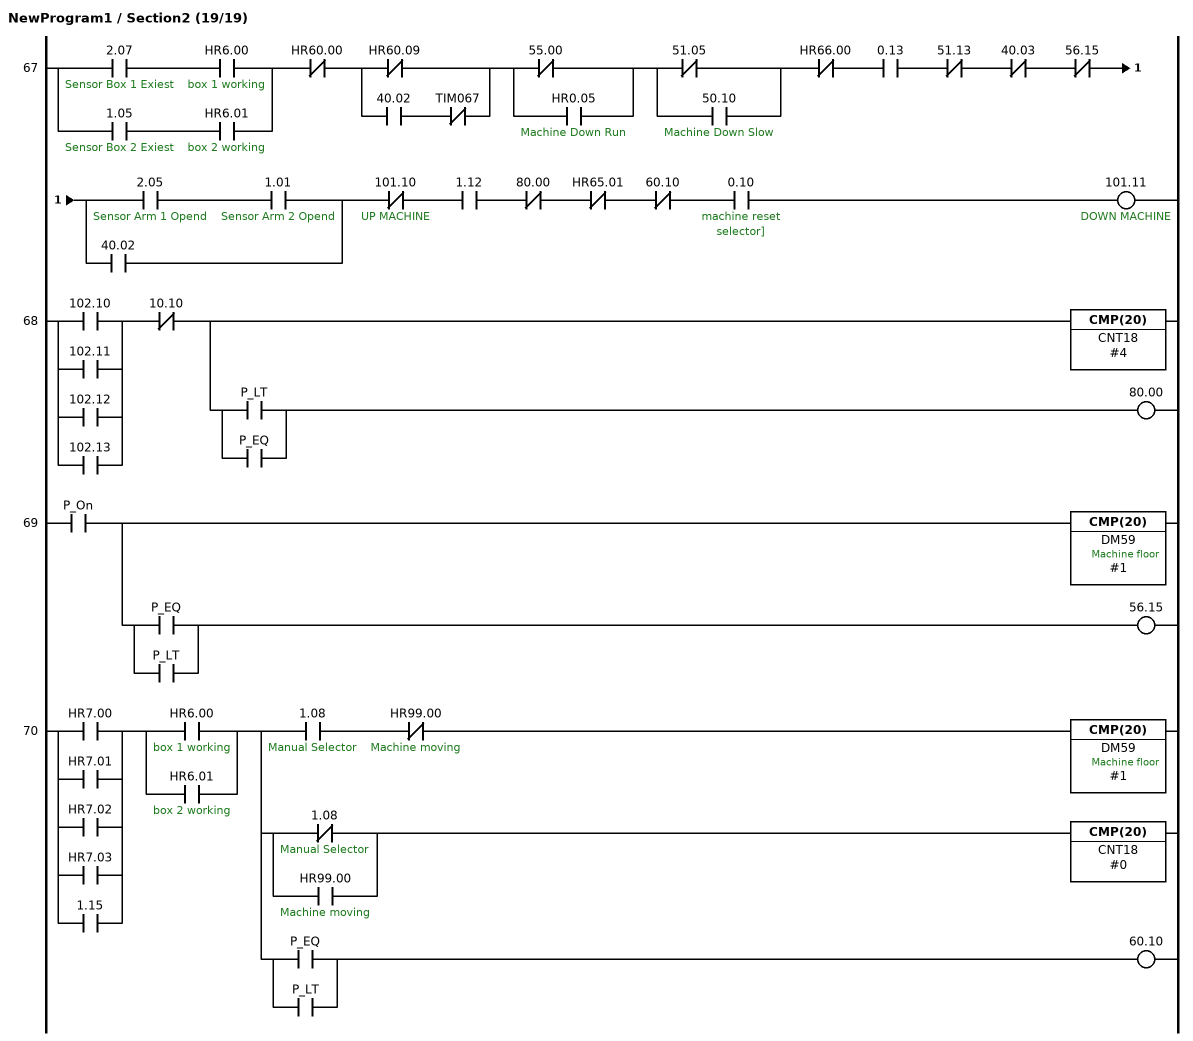
; [picture p24: NewProgram1 / Section2, rungs 67-70]
; rung 67
LD 2.07  ; Sensor Box 1 Exiest
AND HR6.00  ; box 1 working
LD 1.05  ; Sensor Box 2 Exiest
AND HR6.01  ; box 2 working
ORLD
ANDNOT HR60.00
LDNOT HR60.09
LD 40.02
ANDNOT TIM067
ORLD
ANDLD
LDNOT 55.00
OR HR0.05  ; Machine Down Run
ANDLD
LDNOT 51.05
OR 50.10  ; Machine Down Slow
ANDLD
ANDNOT HR66.00
AND 0.13
ANDNOT 51.13
ANDNOT 40.03
ANDNOT 56.15
LD 2.05  ; Sensor Arm 1 Opend
AND 1.01  ; Sensor Arm 2 Opend
OR 40.02
ANDLD
ANDNOT 101.10  ; UP MACHINE
AND 1.12
ANDNOT 80.00
ANDNOT HR65.01
ANDNOT 60.10
AND 0.10  ; machine reset selector]
OUT 101.11  ; DOWN MACHINE
; rung 68
LD 102.10
OR 102.11
OR 102.12
OR 102.13
ANDNOT 10.10
CMP(20) CNT18 #4
LD P_LT
OR P_EQ
ANDLD
OUT 80.00
; rung 69
LD P_On
CMP(20) DM59 #1  ; Machine floor
LD P_EQ
OR P_LT
ANDLD
OUT 56.15
; rung 70
LD HR7.00
OR HR7.01
OR HR7.02
OR HR7.03
OR 1.15
LD HR6.00  ; box 1 working
OR HR6.01  ; box 2 working
ANDLD
OUT TR0
AND 1.08  ; Manual Selector
ANDNOT HR99.00  ; Machine moving
CMP(20) DM59 #1  ; Machine floor
LD TR0
LDNOT 1.08  ; Manual Selector
OR HR99.00  ; Machine moving
ANDLD
CMP(20) CNT18 #0
LD TR0
LD P_EQ
OR P_LT
ANDLD
OUT 60.10

### Section Section3

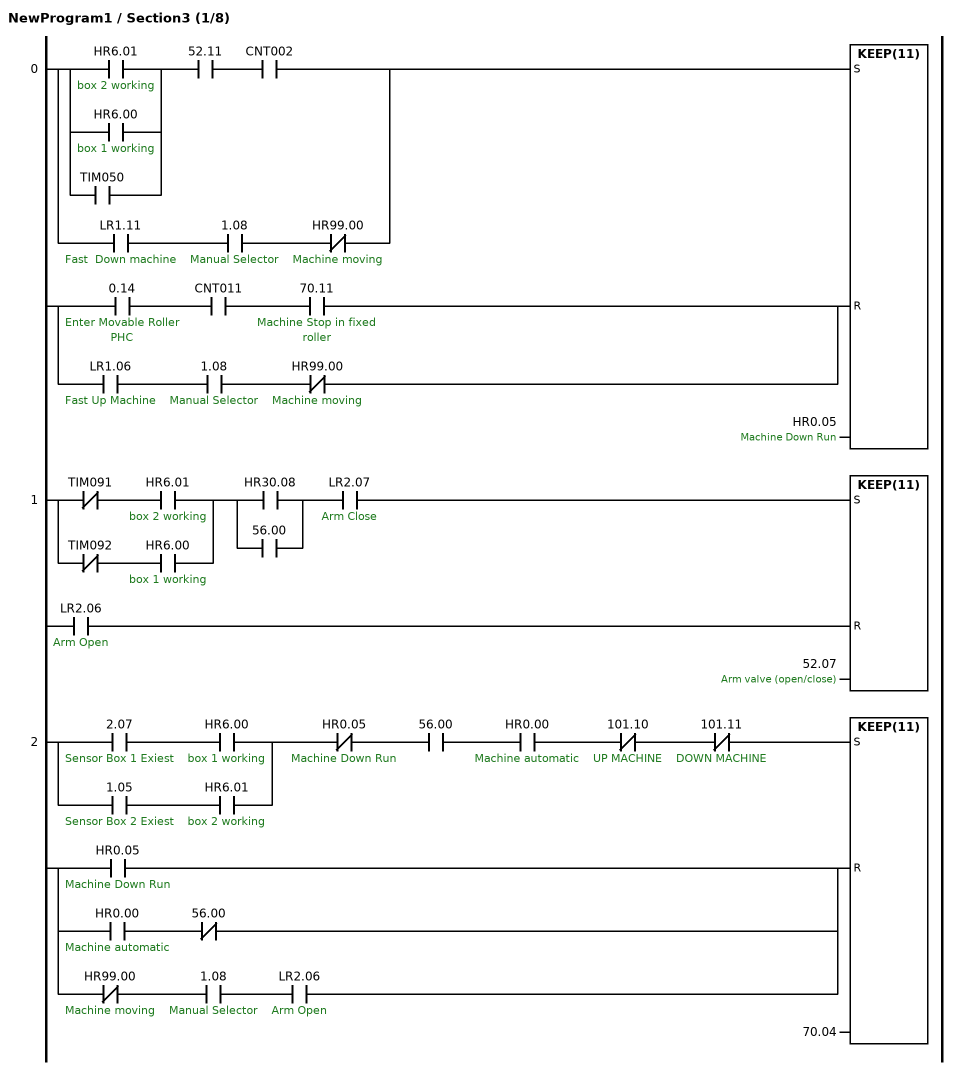
; rung 0
LD HR6.01  ; box 2 working
OR HR6.00  ; box 1 working
OR TIM050
AND 52.11
AND CNT002
LD LR1.11  ; Fast  Down machine
AND 1.08  ; Manual Selector
ANDNOT HR99.00  ; Machine moving
ORLD
LD 0.14  ; Enter Movable Roller PHC
AND CNT011
AND 70.11  ; Machine Stop in fixed roller
LD LR1.06  ; Fast Up Machine
AND 1.08  ; Manual Selector
ANDNOT HR99.00  ; Machine moving
ORLD
KEEP(11) HR0.05  ; Machine Down Run
; rung 1
LDNOT TIM091
AND HR6.01  ; box 2 working
LDNOT TIM092
AND HR6.00  ; box 1 working
ORLD
LD HR30.08
OR 56.00
ANDLD
AND LR2.07  ; Arm Close
LD LR2.06  ; Arm Open
KEEP(11) 52.07  ; Arm valve (open/close)
; rung 2
LD 2.07  ; Sensor Box 1 Exiest
AND HR6.00  ; box 1 working
LD 1.05  ; Sensor Box 2 Exiest
AND HR6.01  ; box 2 working
ORLD
ANDNOT HR0.05  ; Machine Down Run
AND 56.00
AND HR0.00  ; Machine automatic
ANDNOT 101.10  ; UP MACHINE
ANDNOT 101.11  ; DOWN MACHINE
LD HR0.05  ; Machine Down Run
LD HR0.00  ; Machine automatic
ANDNOT 56.00
ORLD
LDNOT HR99.00  ; Machine moving
AND 1.08  ; Manual Selector
AND LR2.06  ; Arm Open
ORLD
KEEP(11) 70.04

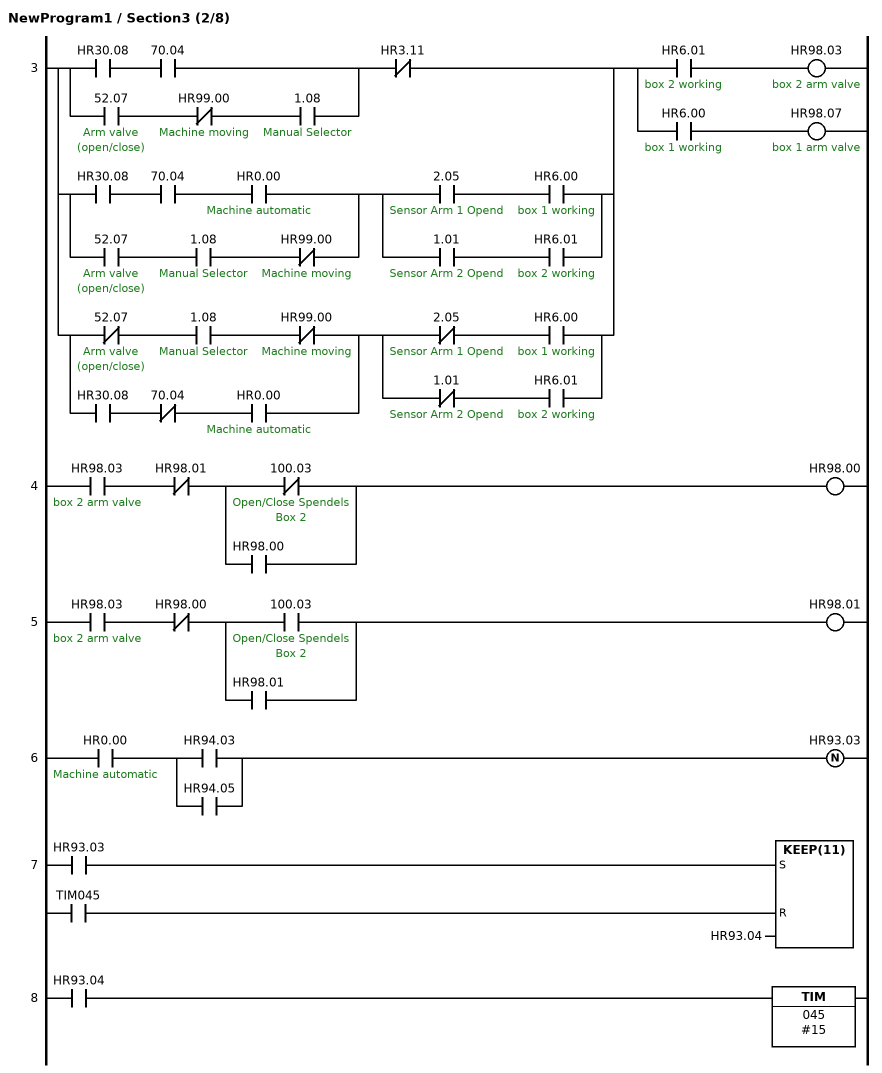
; rung 3
LD HR30.08
AND 70.04
LD 52.07  ; Arm valve (open/close)
ANDNOT HR99.00  ; Machine moving
AND 1.08  ; Manual Selector
ORLD
ANDNOT HR3.11
LD HR30.08
AND 70.04
AND HR0.00  ; Machine automatic
LD 52.07  ; Arm valve (open/close)
AND 1.08  ; Manual Selector
ANDNOT HR99.00  ; Machine moving
ORLD
LD 2.05  ; Sensor Arm 1 Opend
AND HR6.00  ; box 1 working
LD 1.01  ; Sensor Arm 2 Opend
AND HR6.01  ; box 2 working
ORLD
ANDLD
ORLD
LDNOT 52.07  ; Arm valve (open/close)
AND 1.08  ; Manual Selector
ANDNOT HR99.00  ; Machine moving
LD HR30.08
ANDNOT 70.04
AND HR0.00  ; Machine automatic
ORLD
LDNOT 2.05  ; Sensor Arm 1 Opend
AND HR6.00  ; box 1 working
LDNOT 1.01  ; Sensor Arm 2 Opend
AND HR6.01  ; box 2 working
ORLD
ANDLD
ORLD
OUT TR0
AND HR6.01  ; box 2 working
OUT HR98.03  ; box 2 arm valve
LD TR0
AND HR6.00  ; box 1 working
OUT HR98.07  ; box 1 arm valve
; rung 4
LD HR98.03  ; box 2 arm valve
ANDNOT HR98.01
LDNOT 100.03  ; Open/Close Spendels Box 2
OR HR98.00
ANDLD
OUT HR98.00
; rung 5
LD HR98.03  ; box 2 arm valve
ANDNOT HR98.00
LD 100.03  ; Open/Close Spendels Box 2
OR HR98.01
ANDLD
OUT HR98.01
; rung 6
LD HR0.00  ; Machine automatic
LD HR94.03
OR HR94.05
ANDLD
DIFD(14) HR93.03
; rung 7
LD HR93.03
LD TIM045
KEEP(11) HR93.04
; rung 8
LD HR93.04
TIM 045 #15

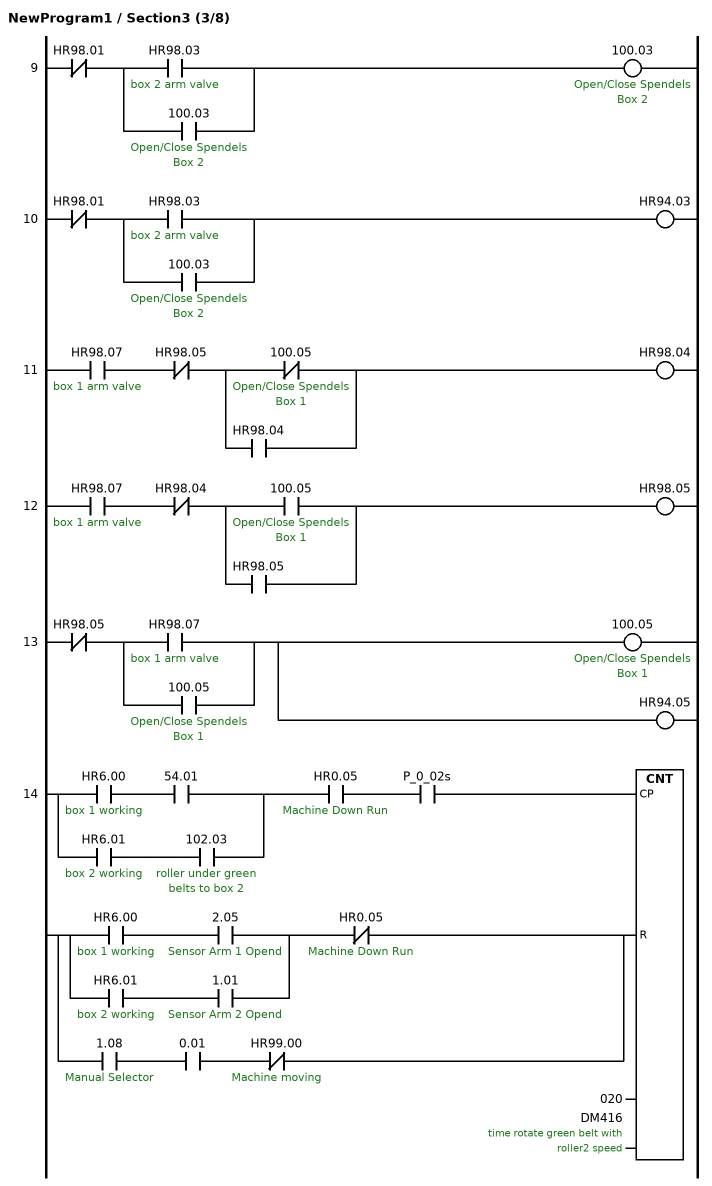
; rung 9
LDNOT HR98.01
LD HR98.03  ; box 2 arm valve
OR 100.03  ; Open/Close Spendels Box 2
ANDLD
OUT 100.03  ; Open/Close Spendels Box 2
; rung 10
LDNOT HR98.01
LD HR98.03  ; box 2 arm valve
OR 100.03  ; Open/Close Spendels Box 2
ANDLD
OUT HR94.03
; rung 11
LD HR98.07  ; box 1 arm valve
ANDNOT HR98.05
LDNOT 100.05  ; Open/Close Spendels Box 1
OR HR98.04
ANDLD
OUT HR98.04
; rung 12
LD HR98.07  ; box 1 arm valve
ANDNOT HR98.04
LD 100.05  ; Open/Close Spendels Box 1
OR HR98.05
ANDLD
OUT HR98.05
; rung 13
LDNOT HR98.05
LD HR98.07  ; box 1 arm valve
OR 100.05  ; Open/Close Spendels Box 1
ANDLD
OUT 100.05  ; Open/Close Spendels Box 1
OUT HR94.05
; rung 14
LD HR6.00  ; box 1 working
AND 54.01
LD HR6.01  ; box 2 working
AND 102.03  ; roller under green belts to box 2
ORLD
AND HR0.05  ; Machine Down Run
AND P_0_02s
LD HR6.00  ; box 1 working
AND 2.05  ; Sensor Arm 1 Opend
LD HR6.01  ; box 2 working
AND 1.01  ; Sensor Arm 2 Opend
ORLD
ANDNOT HR0.05  ; Machine Down Run
LD 1.08  ; Manual Selector
AND 0.01
ANDNOT HR99.00  ; Machine moving
ORLD
CNT 020 DM416  ; time rotate green belt with roller2 speed

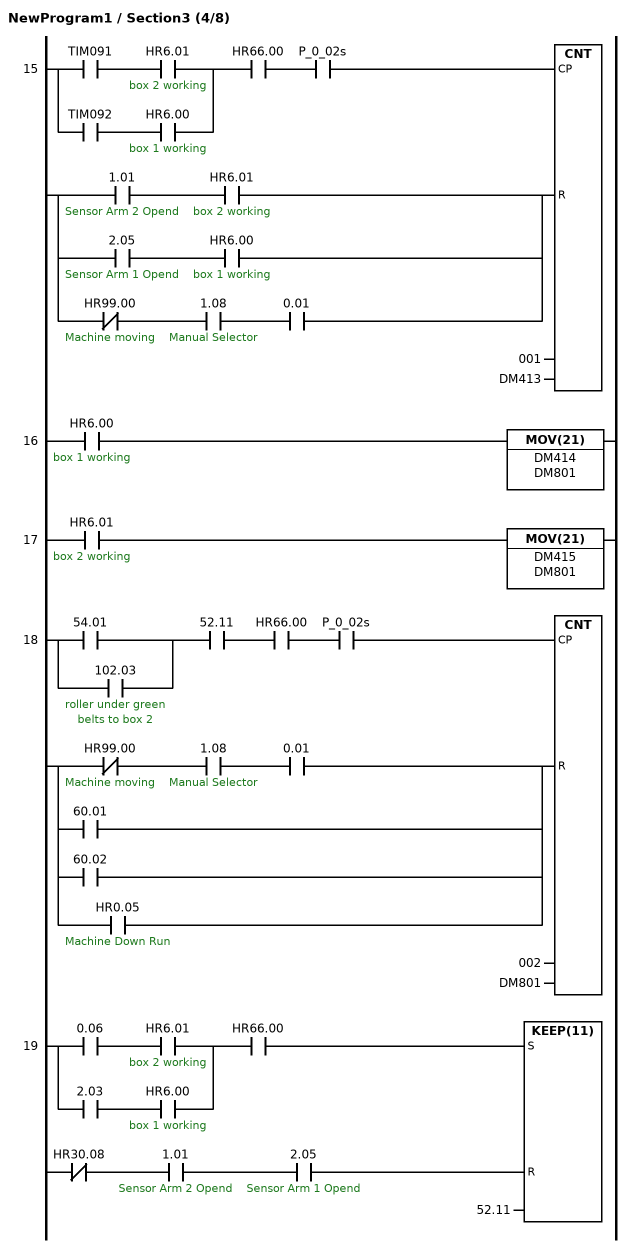
; rung 15
LD TIM091
AND HR6.01  ; box 2 working
LD TIM092
AND HR6.00  ; box 1 working
ORLD
AND HR66.00
AND P_0_02s
LD 1.01  ; Sensor Arm 2 Opend
AND HR6.01  ; box 2 working
LD 2.05  ; Sensor Arm 1 Opend
AND HR6.00  ; box 1 working
ORLD
LDNOT HR99.00  ; Machine moving
AND 1.08  ; Manual Selector
AND 0.01
ORLD
CNT 001 DM413
; rung 16
LD HR6.00  ; box 1 working
MOV(21) DM414 DM801
; rung 17
LD HR6.01  ; box 2 working
MOV(21) DM415 DM801
; rung 18
LD 54.01
OR 102.03  ; roller under green belts to box 2
AND 52.11
AND HR66.00
AND P_0_02s
LDNOT HR99.00  ; Machine moving
AND 1.08  ; Manual Selector
AND 0.01
OR 60.01
OR 60.02
OR HR0.05  ; Machine Down Run
CNT 002 DM801
; rung 19
LD 0.06
AND HR6.01  ; box 2 working
LD 2.03
AND HR6.00  ; box 1 working
ORLD
AND HR66.00
LDNOT HR30.08
AND 1.01  ; Sensor Arm 2 Opend
AND 2.05  ; Sensor Arm 1 Opend
KEEP(11) 52.11

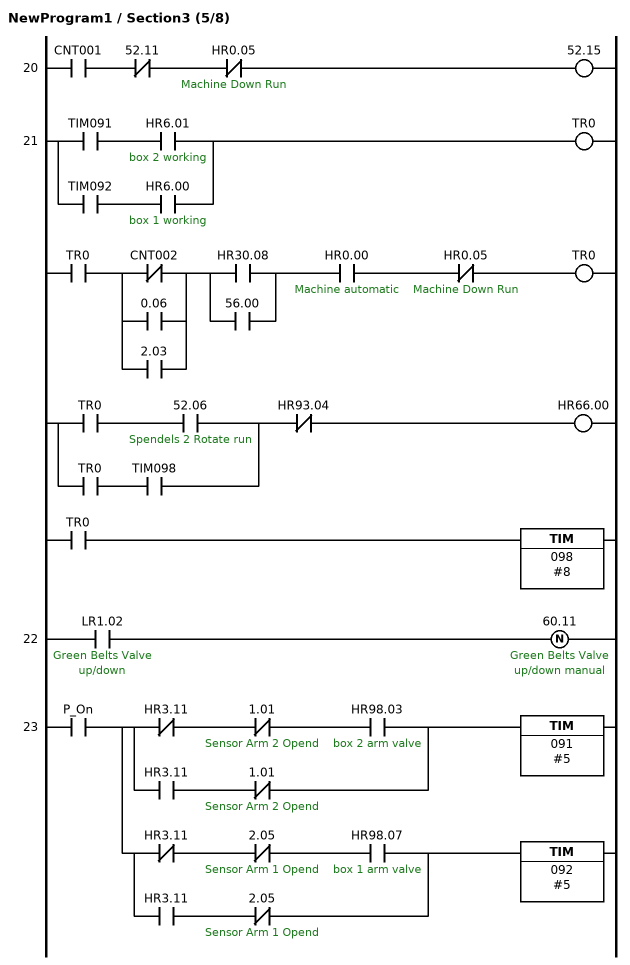
; rung 20
LD CNT001
ANDNOT 52.11
ANDNOT HR0.05  ; Machine Down Run
OUT 52.15
; rung 21
LD TIM091
AND HR6.01  ; box 2 working
LD TIM092
AND HR6.00  ; box 1 working
ORLD
OUT TR0
AND 52.06  ; Spendels 2 Rotate run
LD TR0
LDNOT CNT002
OR 0.06
OR 2.03
ANDLD
LD HR30.08
OR 56.00
ANDLD
AND HR0.00  ; Machine automatic
ANDNOT HR0.05  ; Machine Down Run
OUT TR0
AND TIM098
ORLD
ANDNOT HR93.04
OUT HR66.00
LD TR0
TIM 098 #8
; rung 22
LD LR1.02  ; Green Belts Valve up/down
DIFD(14) 60.11  ; Green Belts Valve up/down manual
; rung 23
LD P_On
OUT TR0
LDNOT HR3.11
ANDNOT 1.01  ; Sensor Arm 2 Opend
AND HR98.03  ; box 2 arm valve
LD HR3.11
ANDNOT 1.01  ; Sensor Arm 2 Opend
ORLD
ANDLD
TIM 091 #5
LD TR0
LDNOT HR3.11
ANDNOT 2.05  ; Sensor Arm 1 Opend
AND HR98.07  ; box 1 arm valve
LD HR3.11
ANDNOT 2.05  ; Sensor Arm 1 Opend
ORLD
ANDLD
TIM 092 #5

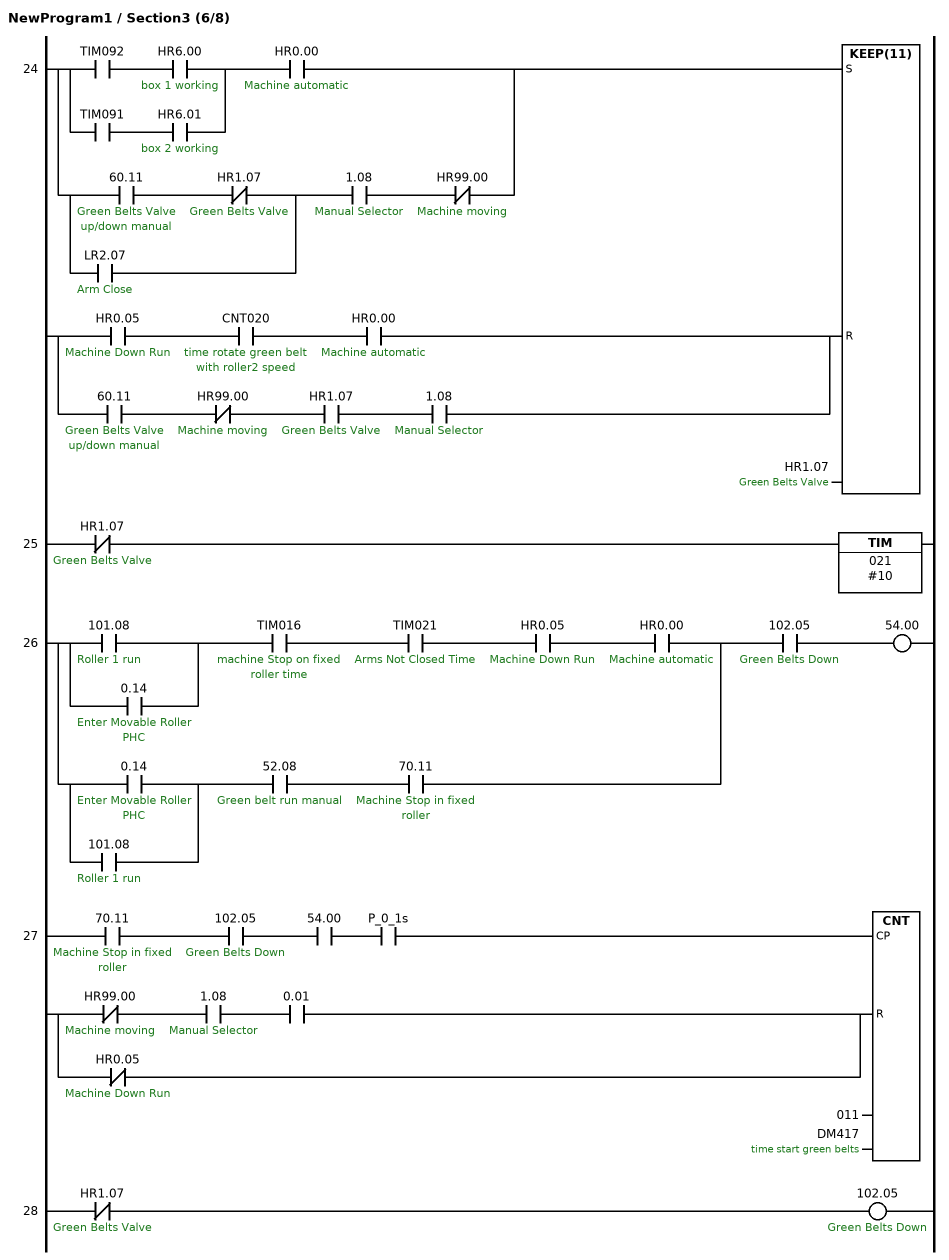
; rung 24
LD TIM092
AND HR6.00  ; box 1 working
LD TIM091
AND HR6.01  ; box 2 working
ORLD
AND HR0.00  ; Machine automatic
LD 60.11  ; Green Belts Valve up/down manual
ANDNOT HR1.07  ; Green Belts Valve
OR LR2.07  ; Arm Close
AND 1.08  ; Manual Selector
ANDNOT HR99.00  ; Machine moving
ORLD
LD HR0.05  ; Machine Down Run
AND CNT020  ; time rotate green belt with roller2 speed
AND HR0.00  ; Machine automatic
LD 60.11  ; Green Belts Valve up/down manual
ANDNOT HR99.00  ; Machine moving
AND HR1.07  ; Green Belts Valve
AND 1.08  ; Manual Selector
ORLD
KEEP(11) HR1.07  ; Green Belts Valve
; rung 25
LDNOT HR1.07  ; Green Belts Valve
TIM 021 #10
; rung 26
LD 101.08  ; Roller 1 run
OR 0.14  ; Enter Movable Roller PHC
AND TIM016  ; machine Stop on fixed roller time
AND TIM021  ; Arms Not Closed Time
AND HR0.05  ; Machine Down Run
AND HR0.00  ; Machine automatic
LD 0.14  ; Enter Movable Roller PHC
OR 101.08  ; Roller 1 run
AND 52.08  ; Green belt run manual
AND 70.11  ; Machine Stop in fixed roller
ORLD
AND 102.05  ; Green Belts Down
OUT 54.00
; rung 27
LD 70.11  ; Machine Stop in fixed roller
AND 102.05  ; Green Belts Down
AND 54.00
AND P_0_1s
LDNOT HR99.00  ; Machine moving
AND 1.08  ; Manual Selector
AND 0.01
ORNOT HR0.05  ; Machine Down Run
CNT 011 DM417  ; time start green belts
; rung 28
LDNOT HR1.07  ; Green Belts Valve
OUT 102.05  ; Green Belts Down

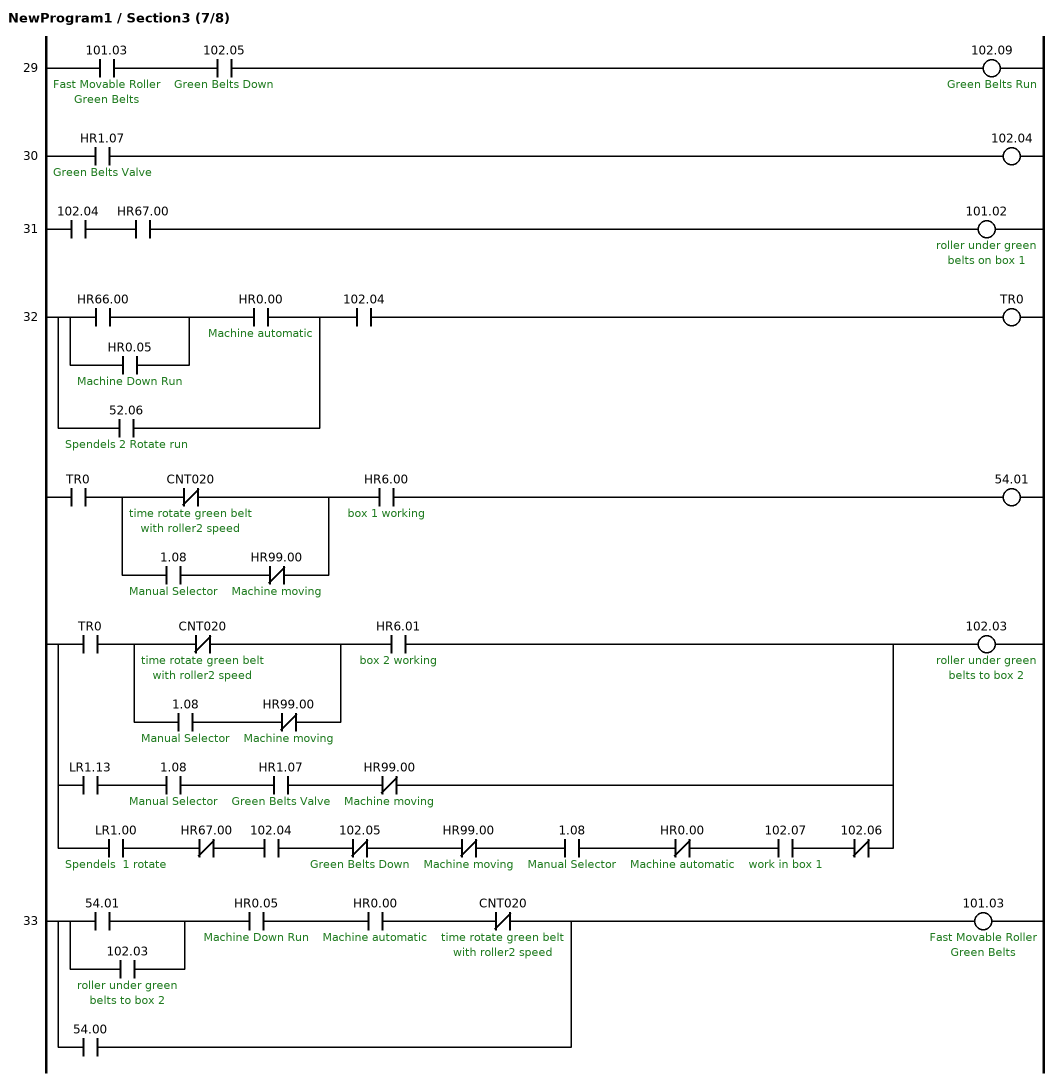
; rung 29
LD 101.03  ; Fast Movable Roller Green Belts
AND 102.05  ; Green Belts Down
OUT 102.09  ; Green Belts Run
; rung 30
LD HR1.07  ; Green Belts Valve
OUT 102.04
; rung 31
LD 102.04
AND HR67.00
OUT 101.02  ; roller under green belts on box 1
; rung 32
LD HR66.00
OR HR0.05  ; Machine Down Run
AND HR0.00  ; Machine automatic
OR 52.06  ; Spendels 2 Rotate run
AND 102.04
OUT TR0
LDNOT CNT020  ; time rotate green belt with roller2 speed
LD 1.08  ; Manual Selector
ANDNOT HR99.00  ; Machine moving
ORLD
ANDLD
AND HR6.00  ; box 1 working
OUT 54.01
LD TR0
LDNOT CNT020  ; time rotate green belt with roller2 speed
LD 1.08  ; Manual Selector
ANDNOT HR99.00  ; Machine moving
ORLD
ANDLD
AND HR6.01  ; box 2 working
LD LR1.13
AND 1.08  ; Manual Selector
AND HR1.07  ; Green Belts Valve
ANDNOT HR99.00  ; Machine moving
LD LR1.00  ; Spendels  1 rotate
ANDNOT HR67.00
AND 102.04
ANDNOT 102.05  ; Green Belts Down
ANDNOT HR99.00  ; Machine moving
AND 1.08  ; Manual Selector
ANDNOT HR0.00  ; Machine automatic
AND 102.07  ; work in box 1
ANDNOT 102.06
ORLD
ORLD
OUT 102.03  ; roller under green belts to box 2
; rung 33
LD 54.01
OR 102.03  ; roller under green belts to box 2
AND HR0.05  ; Machine Down Run
AND HR0.00  ; Machine automatic
ANDNOT CNT020  ; time rotate green belt with roller2 speed
OR 54.00
OUT 101.03  ; Fast Movable Roller Green Belts

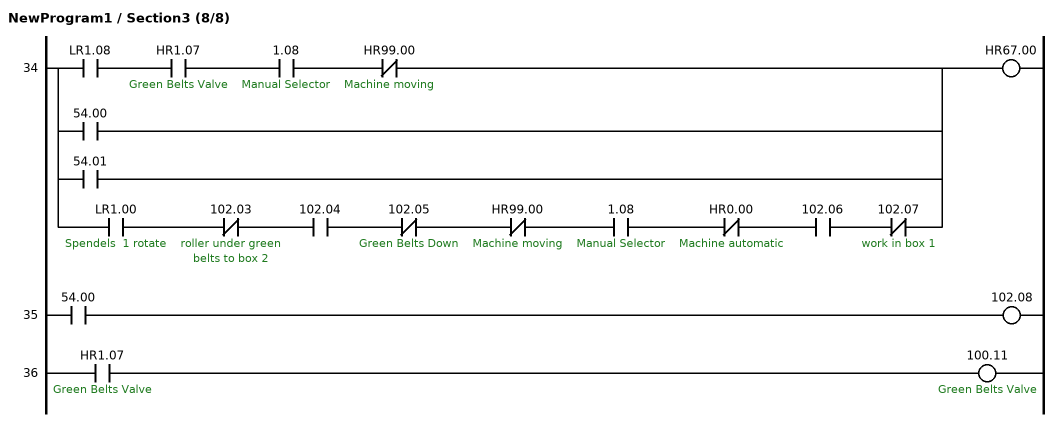
; rung 34
LD LR1.08
AND HR1.07  ; Green Belts Valve
AND 1.08  ; Manual Selector
ANDNOT HR99.00  ; Machine moving
OR 54.00
OR 54.01
LD LR1.00  ; Spendels  1 rotate
ANDNOT 102.03  ; roller under green belts to box 2
AND 102.04
ANDNOT 102.05  ; Green Belts Down
ANDNOT HR99.00  ; Machine moving
AND 1.08  ; Manual Selector
ANDNOT HR0.00  ; Machine automatic
AND 102.06
ANDNOT 102.07  ; work in box 1
ORLD
OUT HR67.00
; rung 35
LD 54.00
OUT 102.08
; rung 36
LD HR1.07  ; Green Belts Valve
OUT 100.11  ; Green Belts Valve

### Section Section4

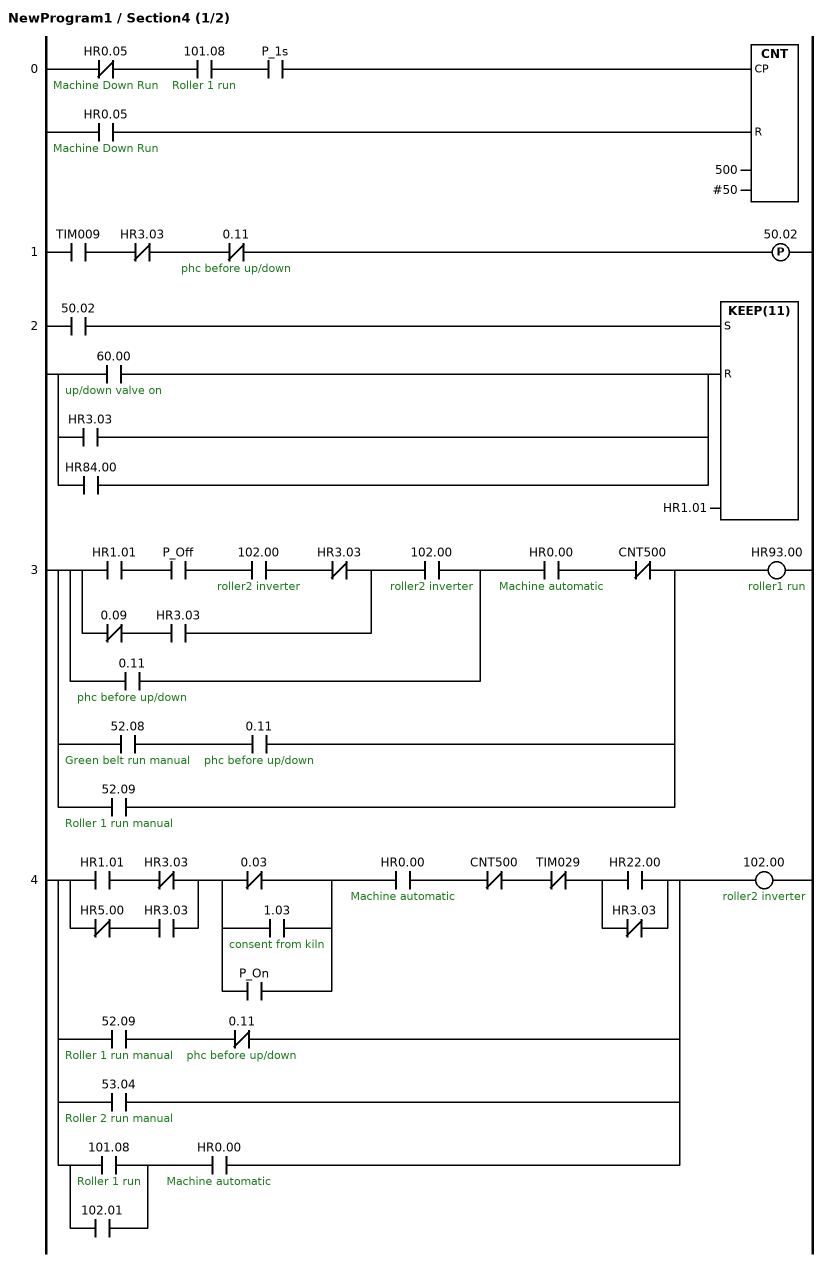
; rung 0
LDNOT HR0.05  ; Machine Down Run
AND 101.08  ; Roller 1 run
AND P_1s
LD HR0.05  ; Machine Down Run
CNT 500 #50
; rung 1
LD TIM009
ANDNOT HR3.03
ANDNOT 0.11  ; phc before up/down
DIFU(13) 50.02
; rung 2
LD 50.02
LD 60.00  ; up/down valve on
OR HR3.03
OR HR84.00
KEEP(11) HR1.01
; rung 3
LD HR1.01
AND P_Off
AND 102.00  ; roller2 inverter
ANDNOT HR3.03
LDNOT 0.09
AND HR3.03
ORLD
AND 102.00  ; roller2 inverter
OR 0.11  ; phc before up/down
AND HR0.00  ; Machine automatic
ANDNOT CNT500
LD 52.08  ; Green belt run manual
AND 0.11  ; phc before up/down
ORLD
OR 52.09  ; Roller 1 run manual
OUT HR93.00  ; roller1 run
; rung 4
LD HR1.01
ANDNOT HR3.03
LDNOT HR5.00
AND HR3.03
ORLD
LDNOT 0.03
OR 1.03  ; consent from kiln
OR P_On
ANDLD
AND HR0.00  ; Machine automatic
ANDNOT CNT500
ANDNOT TIM029
LD HR22.00
ORNOT HR3.03
ANDLD
LD 52.09  ; Roller 1 run manual
ANDNOT 0.11  ; phc before up/down
ORLD
OR 53.04  ; Roller 2 run manual
LD 101.08  ; Roller 1 run
OR 102.01
AND HR0.00  ; Machine automatic
ORLD
OUT 102.00  ; roller2 inverter

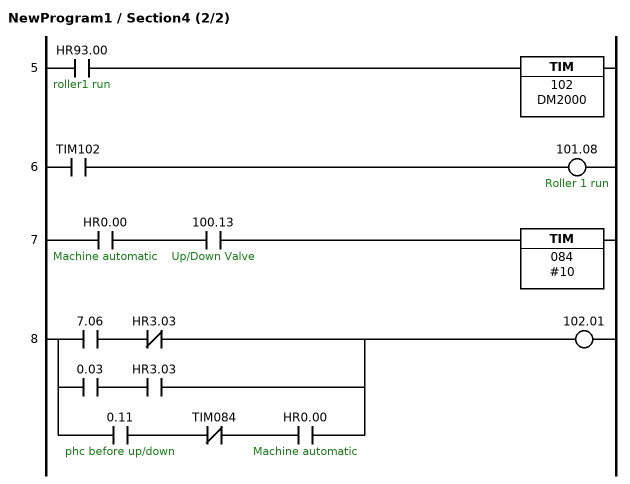
; rung 5
LD HR93.00  ; roller1 run
TIM 102 DM2000
; rung 6
LD TIM102
OUT 101.08  ; Roller 1 run
; rung 7
LD HR0.00  ; Machine automatic
AND 100.13  ; Up/Down Valve
TIM 084 #10
; rung 8
LD 7.06
ANDNOT HR3.03
LD 0.03
AND HR3.03
ORLD
LD 0.11  ; phc before up/down
ANDNOT TIM084
AND HR0.00  ; Machine automatic
ORLD
OUT 102.01

### Section Section5

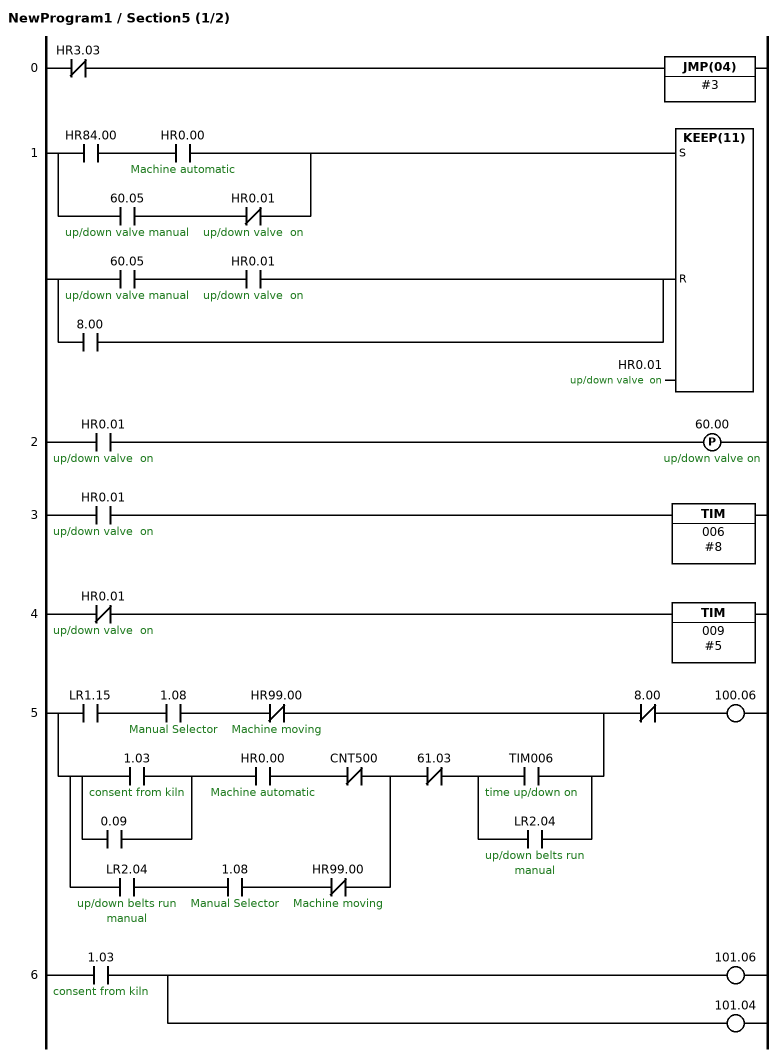
; rung 0
LDNOT HR3.03
JMP(04) #3
; rung 1
LD HR84.00
AND HR0.00  ; Machine automatic
LD 60.05  ; up/down valve manual
ANDNOT HR0.01  ; up/down valve  on
ORLD
LD 60.05  ; up/down valve manual
AND HR0.01  ; up/down valve  on
OR 8.00
KEEP(11) HR0.01  ; up/down valve  on
; rung 2
LD HR0.01  ; up/down valve  on
DIFU(13) 60.00  ; up/down valve on
; rung 3
LD HR0.01  ; up/down valve  on
TIM 006 #8
; rung 4
LDNOT HR0.01  ; up/down valve  on
TIM 009 #5
; rung 5
LD LR1.15
AND 1.08  ; Manual Selector
ANDNOT HR99.00  ; Machine moving
LD 1.03  ; consent from kiln
OR 0.09
AND HR0.00  ; Machine automatic
ANDNOT CNT500
LD LR2.04  ; up/down belts run manual
AND 1.08  ; Manual Selector
ANDNOT HR99.00  ; Machine moving
ORLD
ANDNOT 61.03
LD TIM006  ; time up/down on
OR LR2.04  ; up/down belts run manual
ANDLD
ORLD
ANDNOT 8.00
OUT 100.06
; rung 6
LD 1.03  ; consent from kiln
OUT 101.06
OUT 101.04

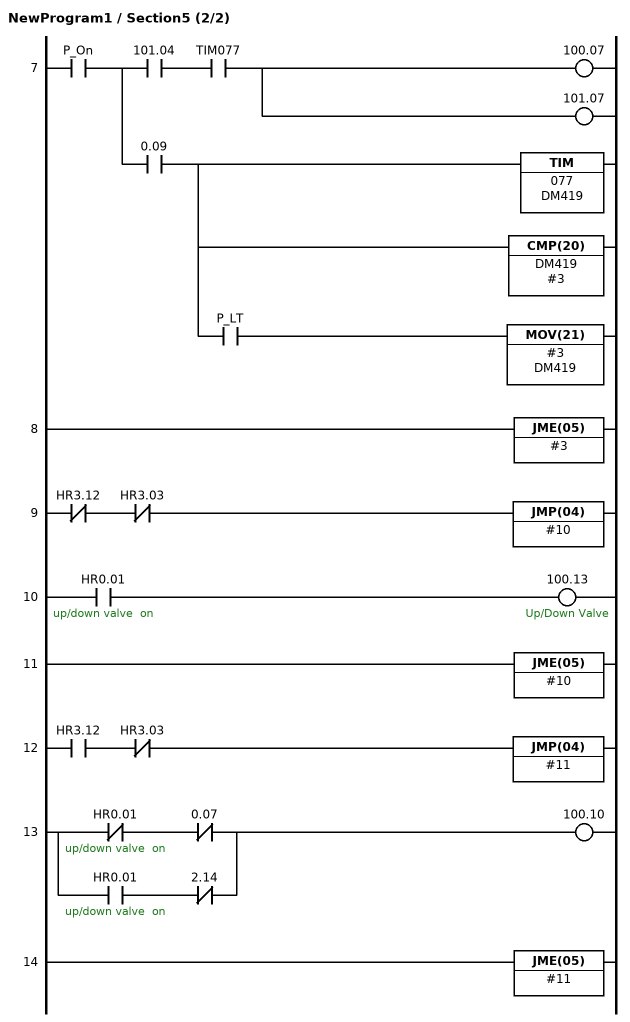
; rung 7
LD P_On
OUT TR0
AND 101.04
AND TIM077
OUT 100.07
OUT 101.07
LD TR0
AND 0.09
TIM 077 DM419
CMP(20) DM419 #3
AND P_LT
MOV(21) #3 DM419
; rung 8
JME(05) #3
; rung 9
LDNOT HR3.12
ANDNOT HR3.03
JMP(04) #10
; rung 10
LD HR0.01  ; up/down valve  on
OUT 100.13  ; Up/Down Valve
; rung 11
JME(05) #10
; rung 12
LD HR3.12
ANDNOT HR3.03
JMP(04) #11
; rung 13
LDNOT HR0.01  ; up/down valve  on
ANDNOT 0.07
LD HR0.01  ; up/down valve  on
ANDNOT 2.14
ORLD
OUT 100.10
; rung 14
JME(05) #11

### Section Section6

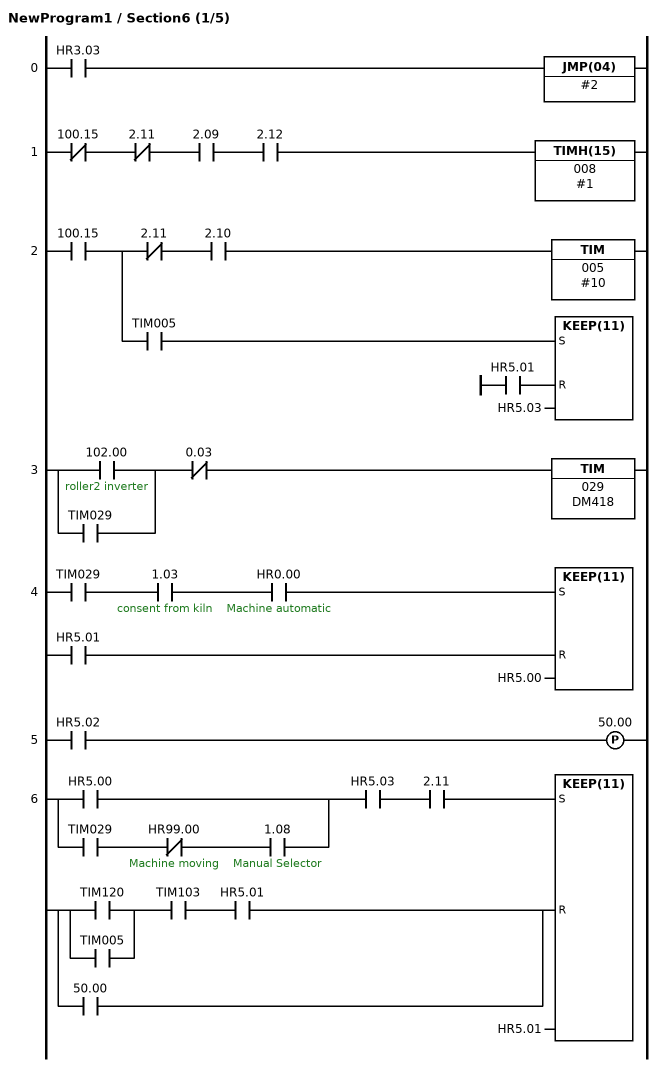
; rung 0
LD HR3.03
JMP(04) #2
; rung 1
LDNOT 100.15
ANDNOT 2.11
AND 2.09
AND 2.12
TIMH(15) 008 #1
; rung 2
LD 100.15
OUT TR0
ANDNOT 2.11
AND 2.10
TIM 005 #10
LD TR0
AND TIM005
LD HR5.01
KEEP(11) HR5.03
; rung 3
LD 102.00  ; roller2 inverter
OR TIM029
ANDNOT 0.03
TIM 029 DM418
; rung 4
LD TIM029
AND 1.03  ; consent from kiln
AND HR0.00  ; Machine automatic
LD HR5.01
KEEP(11) HR5.00
; rung 5
LD HR5.02
DIFU(13) 50.00
; rung 6
LD HR5.00
LD TIM029
ANDNOT HR99.00  ; Machine moving
AND 1.08  ; Manual Selector
ORLD
AND HR5.03
AND 2.11
LD TIM120
OR TIM005
AND TIM103
AND HR5.01
OR 50.00
KEEP(11) HR5.01

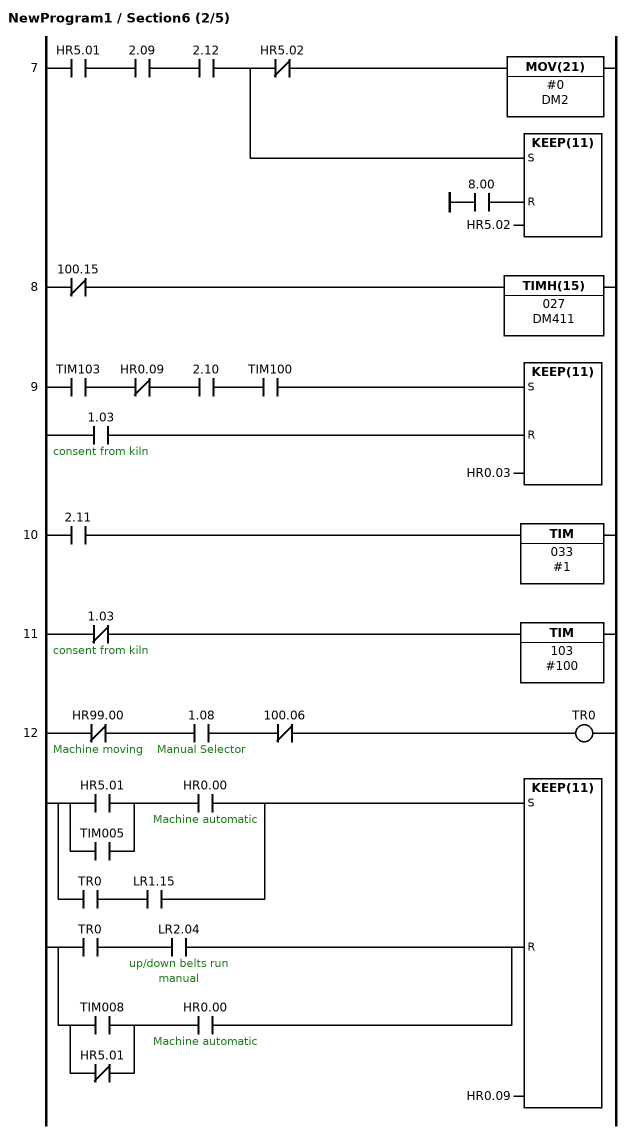
; rung 7
LD HR5.01
AND 2.09
AND 2.12
OUT TR0
ANDNOT HR5.02
MOV(21) #0 DM2
LD TR0
LD 8.00
KEEP(11) HR5.02
; rung 8
LDNOT 100.15
TIMH(15) 027 DM411
; rung 9
LD TIM103
ANDNOT HR0.09
AND 2.10
AND TIM100
LD 1.03  ; consent from kiln
KEEP(11) HR0.03
; rung 10
LD 2.11
TIM 033 #1
; rung 11
LDNOT 1.03  ; consent from kiln
TIM 103 #100
; rung 12
LD HR5.01
OR TIM005
AND HR0.00  ; Machine automatic
LDNOT HR99.00  ; Machine moving
AND 1.08  ; Manual Selector
ANDNOT 100.06
OUT TR0
AND LR1.15
ORLD
LD TR0
AND LR2.04  ; up/down belts run manual
LD TIM008
ORNOT HR5.01
AND HR0.00  ; Machine automatic
ORLD
KEEP(11) HR0.09

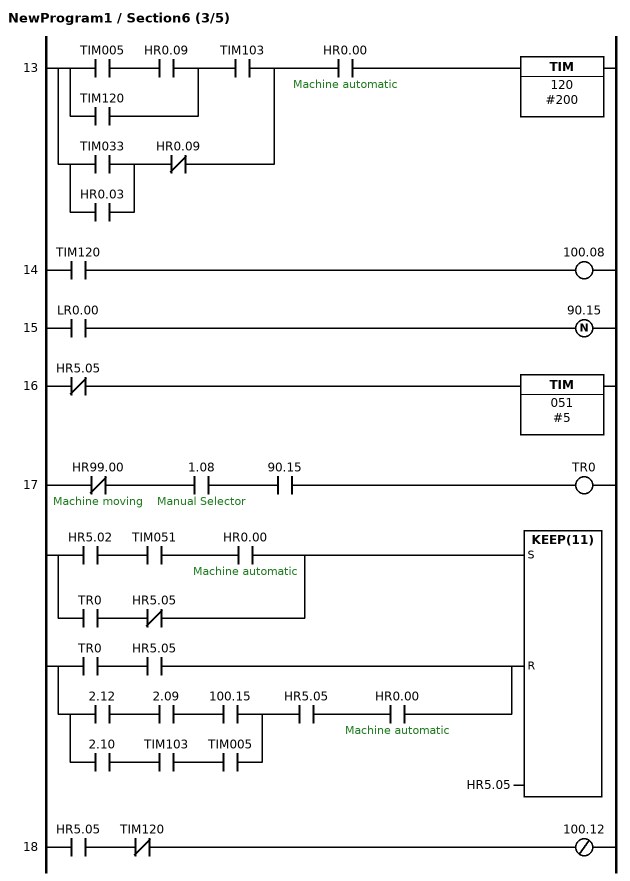
; rung 13
LD TIM005
AND HR0.09
OR TIM120
AND TIM103
LD TIM033
OR HR0.03
ANDNOT HR0.09
ORLD
AND HR0.00  ; Machine automatic
TIM 120 #200
; rung 14
LD TIM120
OUT 100.08
; rung 15
LD LR0.00
DIFD(14) 90.15
; rung 16
LDNOT HR5.05
TIM 051 #5
; rung 17
LD HR5.02
AND TIM051
AND HR0.00  ; Machine automatic
LDNOT HR99.00  ; Machine moving
AND 1.08  ; Manual Selector
AND 90.15
OUT TR0
ANDNOT HR5.05
ORLD
LD TR0
AND HR5.05
LD 2.12
AND 2.09
AND 100.15
LD 2.10
AND TIM103
AND TIM005
ORLD
AND HR5.05
AND HR0.00  ; Machine automatic
ORLD
KEEP(11) HR5.05
; rung 18
LD HR5.05
ANDNOT TIM120
OUTNOT 100.12

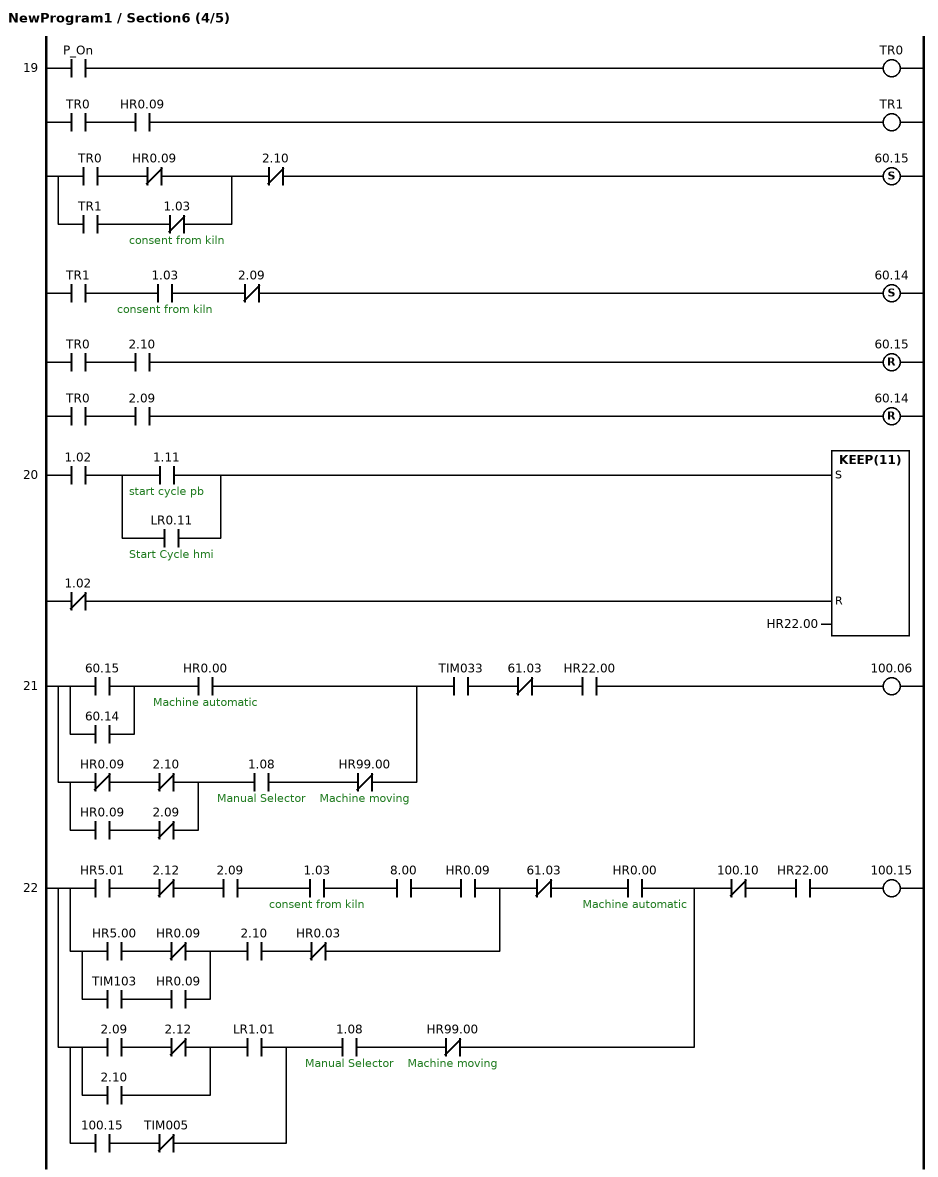
; rung 19
LD P_On
OUT TR0
ANDNOT HR0.09
LD TR0
AND HR0.09
OUT TR1
ANDNOT 1.03  ; consent from kiln
ORLD
ANDNOT 2.10
SET 60.15
LD TR1
AND 1.03  ; consent from kiln
ANDNOT 2.09
SET 60.14
LD TR0
AND 2.10
RSET 60.15
LD TR0
AND 2.09
RSET 60.14
; rung 20
LD 1.02
LD 1.11  ; start cycle pb
OR LR0.11  ; Start Cycle hmi
ANDLD
LDNOT 1.02
KEEP(11) HR22.00
; rung 21
LD 60.15
OR 60.14
AND HR0.00  ; Machine automatic
LDNOT HR0.09
ANDNOT 2.10
LD HR0.09
ANDNOT 2.09
ORLD
AND 1.08  ; Manual Selector
ANDNOT HR99.00  ; Machine moving
ORLD
AND TIM033
ANDNOT 61.03
AND HR22.00
OUT 100.06
; rung 22
LD HR5.01
ANDNOT 2.12
AND 2.09
AND 1.03  ; consent from kiln
AND 8.00
AND HR0.09
LD HR5.00
ANDNOT HR0.09
LD TIM103
AND HR0.09
ORLD
AND 2.10
ANDNOT HR0.03
ORLD
ANDNOT 61.03
AND HR0.00  ; Machine automatic
LD 2.09
ANDNOT 2.12
OR 2.10
AND LR1.01
LD 100.15
ANDNOT TIM005
ORLD
AND 1.08  ; Manual Selector
ANDNOT HR99.00  ; Machine moving
ORLD
ANDNOT 100.10
AND HR22.00
OUT 100.15

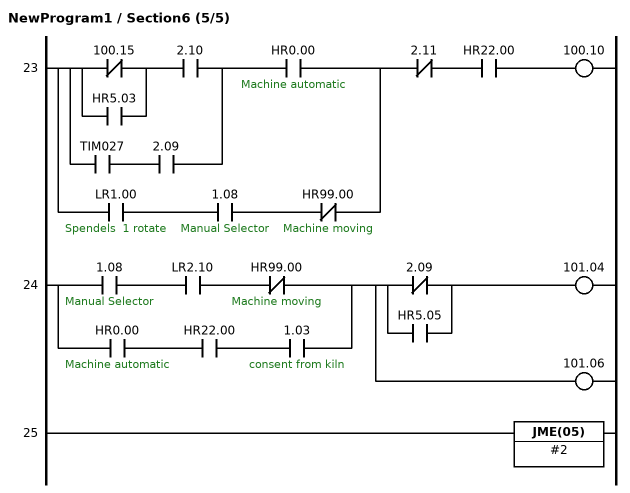
; rung 23
LDNOT 100.15
OR HR5.03
AND 2.10
LD TIM027
AND 2.09
ORLD
AND HR0.00  ; Machine automatic
LD LR1.00  ; Spendels  1 rotate
AND 1.08  ; Manual Selector
ANDNOT HR99.00  ; Machine moving
ORLD
ANDNOT 2.11
AND HR22.00
OUT 100.10
; rung 24
LD 1.08  ; Manual Selector
AND LR2.10
ANDNOT HR99.00  ; Machine moving
LD HR0.00  ; Machine automatic
AND HR22.00
AND 1.03  ; consent from kiln
ORLD
OUT TR0
LDNOT 2.09
OR HR5.05
ANDLD
OUT 101.04
LD TR0
OUT 101.06
; rung 25
JME(05) #2

### Section Section7

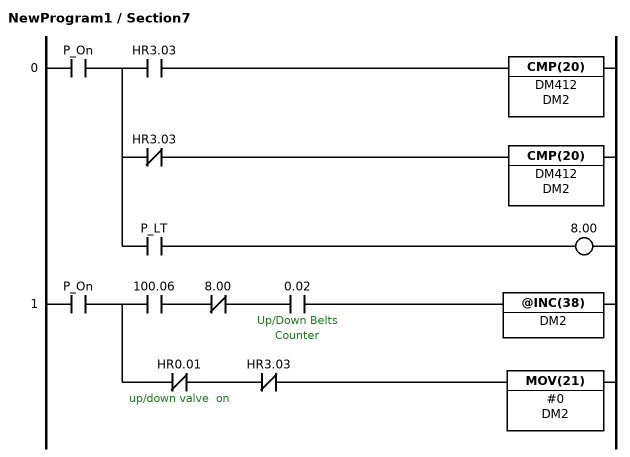
; rung 0
LD P_On
OUT TR0
AND HR3.03
CMP(20) DM412 DM2
LD TR0
ANDNOT HR3.03
CMP(20) DM412 DM2
LD TR0
AND P_LT
OUT 8.00
; rung 1
LD P_On
OUT TR0
AND 100.06
ANDNOT 8.00
AND 0.02  ; Up/Down Belts Counter
@INC(38) DM2
LD TR0
ANDNOT HR0.01  ; up/down valve  on
ANDNOT HR3.03
MOV(21) #0 DM2

### Section Section8

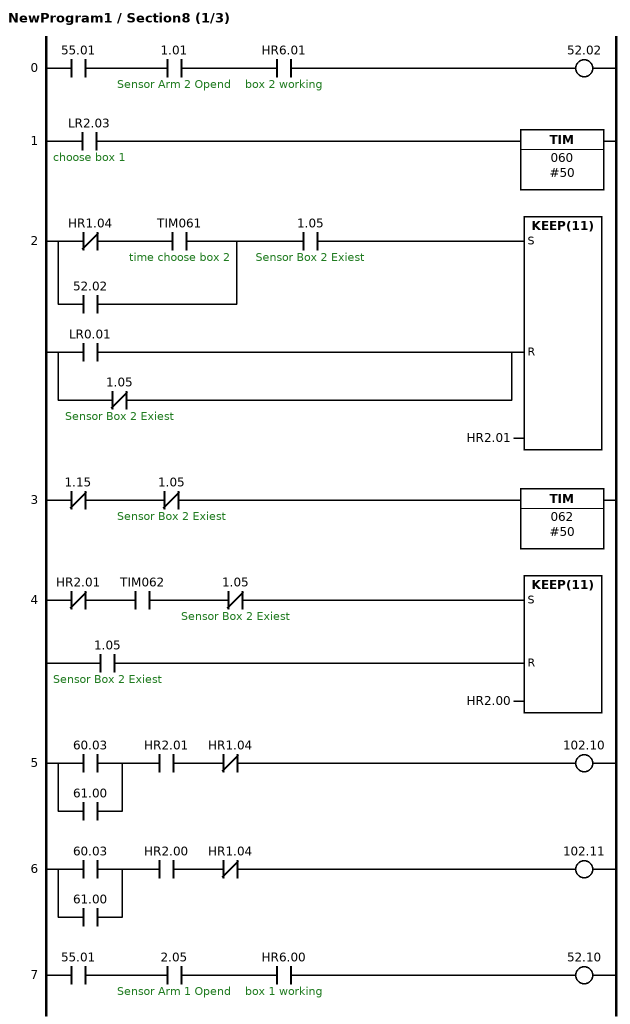
; rung 0
LD 55.01
AND 1.01  ; Sensor Arm 2 Opend
AND HR6.01  ; box 2 working
OUT 52.02
; rung 1
LD LR2.03  ; choose box 1
TIM 060 #50
; rung 2
LDNOT HR1.04
AND TIM061  ; time choose box 2
OR 52.02
AND 1.05  ; Sensor Box 2 Exiest
LD LR0.01
ORNOT 1.05  ; Sensor Box 2 Exiest
KEEP(11) HR2.01
; rung 3
LDNOT 1.15
ANDNOT 1.05  ; Sensor Box 2 Exiest
TIM 062 #50
; rung 4
LDNOT HR2.01
AND TIM062
ANDNOT 1.05  ; Sensor Box 2 Exiest
LD 1.05  ; Sensor Box 2 Exiest
KEEP(11) HR2.00
; rung 5
LD 60.03
OR 61.00
AND HR2.01
ANDNOT HR1.04
OUT 102.10
; rung 6
LD 60.03
OR 61.00
AND HR2.00
ANDNOT HR1.04
OUT 102.11
; rung 7
LD 55.01
AND 2.05  ; Sensor Arm 1 Opend
AND HR6.00  ; box 1 working
OUT 52.10

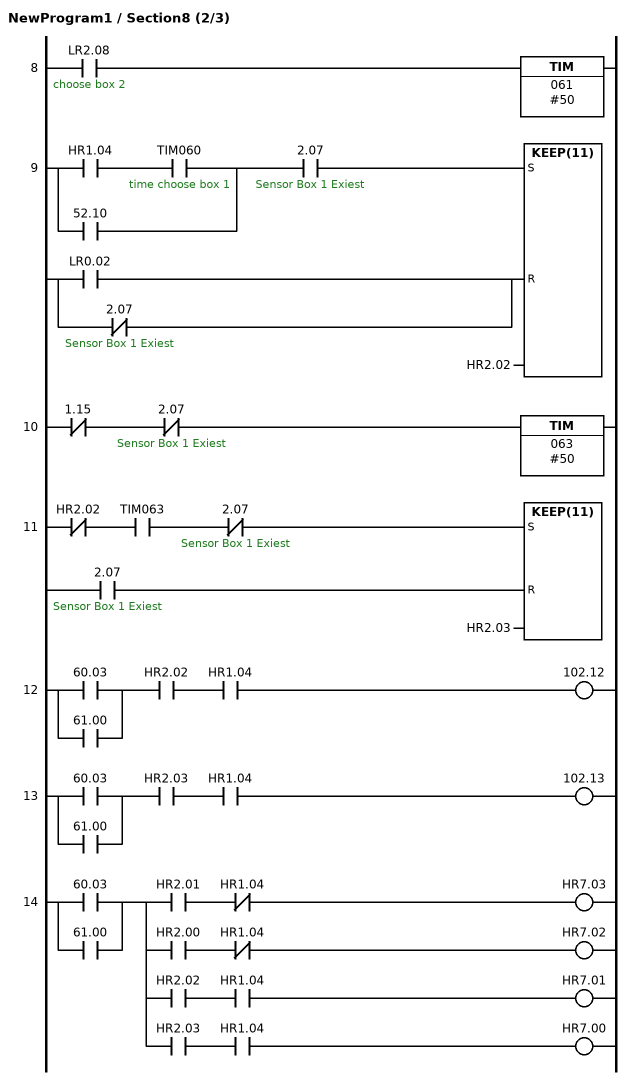
; rung 8
LD LR2.08  ; choose box 2
TIM 061 #50
; rung 9
LD HR1.04
AND TIM060  ; time choose box 1
OR 52.10
AND 2.07  ; Sensor Box 1 Exiest
LD LR0.02
ORNOT 2.07  ; Sensor Box 1 Exiest
KEEP(11) HR2.02
; rung 10
LDNOT 1.15
ANDNOT 2.07  ; Sensor Box 1 Exiest
TIM 063 #50
; rung 11
LDNOT HR2.02
AND TIM063
ANDNOT 2.07  ; Sensor Box 1 Exiest
LD 2.07  ; Sensor Box 1 Exiest
KEEP(11) HR2.03
; rung 12
LD 60.03
OR 61.00
AND HR2.02
AND HR1.04
OUT 102.12
; rung 13
LD 60.03
OR 61.00
AND HR2.03
AND HR1.04
OUT 102.13
; rung 14
LD 60.03
OR 61.00
OUT TR0
AND HR2.01
ANDNOT HR1.04
OUT HR7.03
LD TR0
AND HR2.00
ANDNOT HR1.04
OUT HR7.02
LD TR0
AND HR2.02
AND HR1.04
OUT HR7.01
LD TR0
AND HR2.03
AND HR1.04
OUT HR7.00

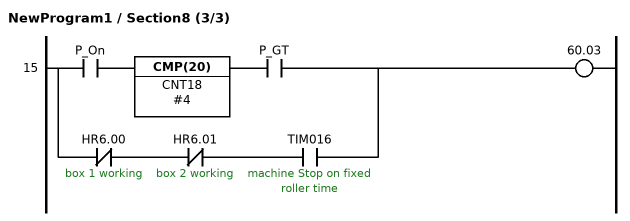
; rung 15
LD P_On
CMP(20) CNT18 #4
AND P_GT
LDNOT HR6.00  ; box 1 working
ANDNOT HR6.01  ; box 2 working
AND TIM016  ; machine Stop on fixed roller time
ORLD
OUT 60.03

### Section Section9

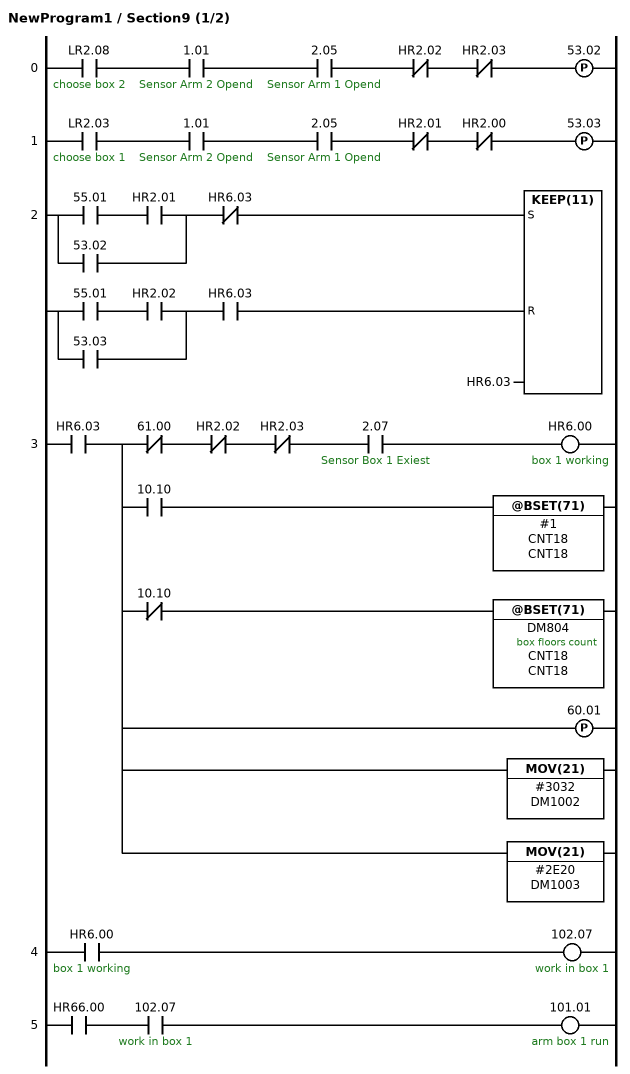
; rung 0
LD LR2.08  ; choose box 2
AND 1.01  ; Sensor Arm 2 Opend
AND 2.05  ; Sensor Arm 1 Opend
ANDNOT HR2.02
ANDNOT HR2.03
DIFU(13) 53.02
; rung 1
LD LR2.03  ; choose box 1
AND 1.01  ; Sensor Arm 2 Opend
AND 2.05  ; Sensor Arm 1 Opend
ANDNOT HR2.01
ANDNOT HR2.00
DIFU(13) 53.03
; rung 2
LD 55.01
AND HR2.01
OR 53.02
ANDNOT HR6.03
LD 55.01
AND HR2.02
OR 53.03
AND HR6.03
KEEP(11) HR6.03
; rung 3
LD HR6.03
OUT TR0
ANDNOT 61.00
ANDNOT HR2.02
ANDNOT HR2.03
AND 2.07  ; Sensor Box 1 Exiest
OUT HR6.00  ; box 1 working
LD TR0
AND 10.10
@BSET(71) #1 CNT18 CNT18
LD TR0
ANDNOT 10.10
@BSET(71) DM804 CNT18 CNT18  ; box floors count
LD TR0
DIFU(13) 60.01
MOV(21) #3032 DM1002
MOV(21) #2E20 DM1003
; rung 4
LD HR6.00  ; box 1 working
OUT 102.07  ; work in box 1
; rung 5
LD HR66.00
AND 102.07  ; work in box 1
OUT 101.01  ; arm box 1 run

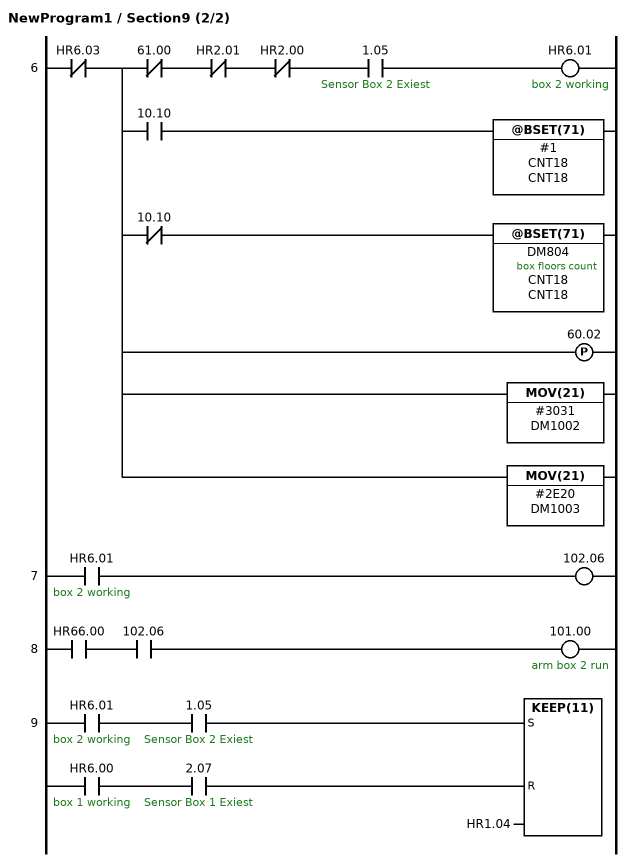
; rung 6
LDNOT HR6.03
OUT TR0
ANDNOT 61.00
ANDNOT HR2.01
ANDNOT HR2.00
AND 1.05  ; Sensor Box 2 Exiest
OUT HR6.01  ; box 2 working
LD TR0
AND 10.10
@BSET(71) #1 CNT18 CNT18
LD TR0
ANDNOT 10.10
@BSET(71) DM804 CNT18 CNT18  ; box floors count
LD TR0
DIFU(13) 60.02
MOV(21) #3031 DM1002
MOV(21) #2E20 DM1003
; rung 7
LD HR6.01  ; box 2 working
OUT 102.06
; rung 8
LD HR66.00
AND 102.06
OUT 101.00  ; arm box 2 run
; rung 9
LD HR6.01  ; box 2 working
AND 1.05  ; Sensor Box 2 Exiest
LD HR6.00  ; box 1 working
AND 2.07  ; Sensor Box 1 Exiest
KEEP(11) HR1.04

### Section Section10

